(* IEC 61131-3 sources: ml2plc/benchmarks/st (part 17) *)

(* ---- MLP8_straton.st ---- *)
FUNCTION_BLOCK MLP8_FB

    (* Model Inputs/Outputs *)
VAR_INPUT
    input_data : REAL;
END_VAR

VAR_OUTPUT
    output_data : ARRAY[0..2] OF REAL;
END_VAR

VAR
    CONSTANT weights_0 : ARRAY[0..63] OF REAL := [0.566726267, 0.697450101, 0.648469865, -0.244775116, -0.237901151, 0.738550067, 0.472831041, 0.688409746, -0.0405910909, 0.54798907, 0.658046842, 0.487694085, 0.466130763, -0.209909201, -0.167861477, -0.185364306, -0.119988531, 0.702987075, 0.664516151, 0.492332131, 0.366119206, -0.231371135, 0.561849892, -0.299611568, 0.524393439, -0.0369002223, -0.225777417, 0.425555229, 0.708118021, 0.6373595, -0.302317858, 0.514846981, -0.277802587, -0.160284445, -0.23097758, 0.685079992, -0.0133622587, -0.197633862, 0.646109998, -0.0195143819, -0.00467607379, 0.46406725, -0.240666151, 0.522509336, -0.235457808, 0.497557789, -0.176456973, 0.530339539, -0.191211104, 0.541193664, 0.750494003, -0.0375860631, -0.214687645, -0.243620768, 0.659598589, 0.568989158, -0.3036699, 0.672104239, -0.244726226, 0.594575703, 0.681357145, -0.109698236, -0.107163459, 0.571734607];
    CONSTANT bias_0 : ARRAY[0..63] OF REAL := [-0.127067611, -0.150965586, -0.145847186, 0, 0, -0.142355159, 0.536983192, -0.151563853, 0, -0.108020559, 0.215985522, -0.109748609, -0.104939878, 0, 0, 0, 0, -0.15642038, -0.148533463, -0.110406905, 0.563737273, 0, -0.111798488, 0, -0.114780053, 0, 0, -0.0961699262, -0.133371383, -0.128657907, 0, -0.115175709, 0, 0, 0, -0.153447583, 0, 0, -0.0991757438, 0, 0, -0.103414647, 0, -0.117680125, 0, -0.111900046, 0, -0.119580522, 0, -0.121857166, -0.127358705, 0, 0, 0, -0.138788998, -0.125557691, 0, -0.147434101, 0, -0.126147434, -0.151844159, 0, 0, -0.126771837];
    CONSTANT weights_1 : ARRAY[0..3071] OF REAL := [-0.508529365, 0.777783334, -0.589114606, 0.647827327, -0.879598022, 0.374501675, -0.233010441, 0.470010132, 0.398335785, -0.835246623, -0.883157551, 0.755935609, -0.212538779, -0.178419977, 0.952007294, -0.811082065, 0.467197567, -0.294056267, -0.467858523, 1.01234376, 0.25377509, 0.712045431, -0.0497531593, -0.882072449, -0.987796485, 0.161702394, 0.587665379, 0.0541041195, 0.0643232763, 0.158115536, -0.557613134, -0.822882295, -0.602058291, -0.260582656, -1.05500817, -0.0198417753, 0.0395283103, 0.0372411311, 0.594341755, 0.584856927, 0.0607305169, -0.298460275, -0.480308563, 0.551810563, -0.737427711, 0.145618647, -0.499337137, -0.307826608, -0.473668456, 0.347774506, -0.187618226, 0.751432717, -0.689023435, 0.527891994, -0.193951294, 0.760585308, 0.328736782, -0.449620336, -0.498079717, 0.947781801, 0.0636215508, 0.190816671, 0.423609227, -0.963524342, 0.335212857, -0.300242186, -0.496480465, 0.62573868, 0.376674086, 0.36957857, 0.273251772, -0.723223269, -0.979038298, -0.128652185, 0.820281744, -0.150052547, -0.043580249, -0.184555292, -0.590572476, -1.00735581, -0.268060088, -0.245665103, -0.599425495, -0.135427296, -0.0110698044, -0.163606152, 0.57665354, 0.615970254, 0.0755210519, -0.242924631, -0.371946365, 0.521858156, -0.288352877, -0.214046448, -0.42009899, -0.499587744, -0.819006622, 0.522933841, -0.480003029, 0.688604951, -0.966424167, 0.622771263, -0.0291726999, 0.808974981, 0.633017004, -0.567950785, -0.715922832, 0.645944357, 0.126155347, 0.0951944366, 0.545724213, -0.931986749, 0.160165772, -0.0631896481, -0.52388972, 0.583337784, 0.470121413, 0.267368495, -0.0256699882, -1.1038264, -1.04683483, -0.0606382638, 0.849855661, 0.0996483564, -0.0824714303, 0.0362196565, -0.66673249, -1.04458475, -0.338297427, -0.53378427, -0.989768386, -0.225421071, 0.0280500948, 0.0889418721, 0.467521846, 0.709094465, 0.224540606, -0.255299211, -0.531706095, 0.613625348, -0.721871734, -0.14013961, -0.32255891, -0.276349634, -0.0558475852, -0.0150698572, 0.189445347, -0.224641621, 0.0600843728, -0.199145943, -0.114447266, 0.0321756005, -0.0139652044, 0.139568895, -0.136456579, 0.0218596458, 0.191010177, -0.0243975371, 0.0602264702, 0.0723614395, -0.0896188021, -0.058872506, 0.106127173, 0.0416764319, -0.0183494538, -0.199132025, 0.223530114, 0.00858539343, 0.0776902437, 0.0439737141, 0.00252109766, -0.226854458, 0.0800455809, 0.216010183, 0.174708903, -0.132116258, 0.0539589822, 0.0233850181, 0.126452208, 0.0195031166, 0.20596543, 0.0608135164, 0.0942558348, 0.22737518, -0.0990859717, -0.0777076781, -0.00981768966, -0.229763716, 0.0728095174, -0.208888695, -0.0588912666, 0.00719544291, -0.0642014891, 0.208572537, 0.185866833, -0.205061138, -0.190968722, -0.0123857558, 0.0851061344, 0.0569832623, 0.182903767, -0.165526241, -0.17117624, 0.0841451287, -0.178321734, -0.0988931656, 0.21516645, 0.203568548, -0.0786485076, 0.102775037, 0.104268342, 0.15373078, 0.23019889, 0.0220953524, -0.00975424051, 0.0953029096, -0.223771766, 0.229721338, -0.0257629901, 0.179429203, 0.0443455875, 0.191467524, 0.143349111, 0.21192956, 0.0171111971, -0.0315240026, 0.0892953277, -0.0647144169, -0.176158011, -0.0644855201, -0.15905486, -0.0899337977, 0.0437249541, 0.0412196219, -0.0510214269, -0.103800446, 0.0931487083, 0.183442682, 0.187456101, 0.18982622, -0.630144417, 0.611605942, -0.276451319, 0.63561976, -0.841786385, 0.105425507, 0.118410617, 0.642714441, 0.30139786, -0.423010617, -0.160331935, 0.631173253, -0.0531943738, 0.0132380854, 0.557571173, -0.680383444, 0.229302496, -0.0644649342, -0.597031713, 0.604079127, 0.0652358979, 0.508375168, 0.192985371, -0.684397638, -0.757217824, -0.0915823877, 0.624771178, 0.073392421, -0.213347048, -0.0439970493, -0.179815233, -0.822682321, -0.290968657, -0.449465156, -0.282994241, 0.0222680271, 0.202416599, 0.0366479158, 0.648888052, 0.345080584, -0.0183112063, -0.057644885, -0.33952108, 0.505236089, -0.269680262, 0.0832733512, -0.367935091, -0.27335614, 0.407757968, 0.238256618, 0.34742102, 0.0945411921, 0.179025948, -0.160453767, 0.0919690207, -0.0016620002, -0.140238672, 0.610232711, 0.662595987, 0.403355569, -0.108785428, 0.0517903045, 0.435860395, -0.0251670647, -0.251344532, 0.452141792, 0.557143986, 0.458476484, -0.255402505, 0.175111428, 0.455911607, 0.412472844, 0.218193471, -0.207911894, 0.0693136305, -0.059445411, -0.169521675, -0.182679832, 0.519502401, -0.0549139269, 0.497394502, 0.420575768, 0.255482435, -0.0491585582, 0.042904973, -0.192346439, 0.095114693, -0.346379042, -0.0267166235, 0.220421061, 0.3648085, -0.321888626, 0.446793377, -0.0310783982, 0.233682126, 0.388623834, -0.583991706, 0.505147576, -0.534565687, 0.322568089, -1.03081346, 0.283099979, 0.194360659, 0.706190765, 0.641339362, -0.426852167, -0.447203308, 0.554000199, 0.0497648604, 0.123939805, 0.853530824, -1.04427862, 0.252899885, -0.233157471, -0.306790262, 0.776063979, 0.559772849, 0.542160273, 0.0403436981, -1.10041475, -1.00884628, -0.138749599, 0.702059388, 0.0610145628, -0.0819382966, -0.111110725, -0.482868969, -0.934108913, -0.362628788, -0.359785378, -0.733438969, -0.060155347, -0.0659447312, 0.201255053, 0.359661549, 0.509634912, -0.0411985293, -0.504819214, -0.286087692, 0.544379532, -0.52835089, -0.0581299067, -0.380262613, -0.474460214, 0.0785628557, 0.193065852, -0.0540531427, 0.0867037475, -0.0140087456, -0.159107059, 0.16856578, 0.114497095, 0.0728079677, 0.123832315, 0.134191304, 0.201696187, -0.141746759, 0.213595003, -0.2263944, 0.0249090195, -0.158394754, -0.0716763884, 0.152066469, 0.0486070514, 0.111786395, 0.0807827115, 0.0409047008, 0.220125973, -0.219644442, 0.0905397534, 0.202887952, -0.153925478, -0.0712448508, 0.224727035, 0.116824895, 0.211984366, 0.0860830545, 0.134800911, -0.038962245, -0.0824456513, 0.0818852186, -0.0403479487, 0.0376374722, -0.108327284, 0.0718497038, 0.216866136, -0.213927254, 0.0031440109, -0.0106695592, -0.0465998203, -0.195866793, -0.214657992, -0.44059667, 0.660695314, -0.367561132, 0.594573438, -0.827821732, 0.38140139, -0.109366305, 0.564865768, 0.398382038, -0.642758369, -0.504486442, 0.811359286, 0.0293445885, -0.0519628488, 0.806313336, -0.863483965, 0.288089395, -0.143644974, -0.205591589, 0.838227034, 0.285395503, 0.240181088, 0.432383686, -0.649837255, -0.91485858, -0.177318007, 0.784425735, 0.22021389, 0.192846447, -0.0329939127, -0.348731846, -0.652700245, -0.339493215, -0.16938825, -0.534539282, 0.181898445, 0.178422064, -0.0549968779, 0.344090849, 0.254576117, -0.172308087, -0.139661431, -0.249803483, 0.395636946, -0.541676044, 0.201305479, -0.331647396, -0.306729645, 0.404410243, 0.250662118, 0.147280648, 0.502067685, 0.137784511, 0.0780866221, 0.0449218713, 0.323366255, 0.0272866227, 0.0769802928, -0.00688272109, 0.454549521, -0.147471949, -0.0136137269, 0.257623971, 0.0870388225, 0.0359390229, 0.164906204, 0.0806759894, 0.18752256, 0.211298063, 0.36549443, 0.381839573, 0.0227036048, 0.056207899, -0.0421615988, 0.497502565, 0.047046423, 0.209912181, 0.0365511775, 0.0822928399, 0.0565427281, 0.17033419, 0.133746162, -0.0657917038, -0.102406234, -0.0849392116, 0.171123147, 0.401582569, -0.0835181177, -0.133074522, 0.38805151, 0.281278849, 0.0756753385, 0.273700088, -0.114257708, 0.322280556, 0.240192294, -0.459217519, 0.901713192, -0.382146418, 0.67524451, -0.830624104, 0.424378633, -0.190720469, 0.905839324, 0.637098491, -0.503638327, -0.900598824, 1.19751096, 0.00358029734, -0.237770662, 1.01180136, -0.902854562, 0.475136936, -0.206849128, -0.774593174, 1.03993857, 0.640500665, 0.510213614, 0.0561259016, -1.24519598, -1.01733959, -0.115967944, 0.81452024, -0.161395952, -0.0437688082, -0.156050742, -0.53688693, -1.06002426, -0.470631003, -0.52531755, -1.12388718, 0.208761662, -0.176574588, -0.214394152, 0.646233439, 0.506878614, -0.0175239854, -0.63169241, -0.766251266, 0.681717753, -0.629178941, 0.117619962, -0.785952628, -0.735168219, -0.948679447, 0.878256857, -0.590300083, 1.04297566, -0.968591094, 0.856882274, 0.0444319323, 0.841967404, 0.672772825, -0.959409237, -0.734882236, 1.03502762, -0.0881304815, 0.137461543, 0.820007682, -1.38987863, 0.50563246, -0.212394595, -0.653115332, 1.03907979, 0.750977933, 0.649298608, -0.129806831, -1.40875912, -1.13032782, 0.180365622, 0.864530802, -0.155418515, -0.00242756307, -0.212027237, -0.488034099, -1.3115921, -0.619424522, -0.484913111, -1.09705448, -0.128922701, -0.13195011, -0.180079982, 1.18086195, 0.745139778, 0.167641819, -0.668225586, -0.77761519, 0.425894529, -0.626781106, -0.18818298, -0.721377492, -0.526926816, 0.215941429, -0.123659819, -0.184358388, 0.043376863, -0.0120955408, 0.122474253, -0.0583063215, -0.212231085, 0.183268249, 0.0962251723, -0.147334784, -0.11822731, 0.0362046957, 0.0269062817, -0.194129512, 0.0830053687, -0.161627054, -0.0567752719, -0.145187616, 0.120651454, -0.0233496577, 0.206467032, -0.17806983, -0.0681224167, 0.104563296, -0.218612805, 0.0865324736, 0.0349574983, -0.0137506574, 0.134827524, -0.0367743969, 0.184188545, 0.197318703, -0.0225695372, -0.221328974, -0.0929350406, -0.177381575, 0.00736005604, 0.037692219, 0.000573635101, 0.0186697245, -0.0238907337, -0.177731991, -0.129223391, 0.0824308693, -0.200551838, -0.16154848, 0.199765205, 0.206477582, 0.101242274, 0.0433039069, 0.0258513987, 0.160764426, -0.0691497177, -0.084734261, 0.227003336, -0.125068694, 0.146611392, -0.00917938352, -0.168416351, 0.136403561, -0.189610675, -0.127061039, 0.00317269564, 0.201314688, -0.0198562294, -0.144739896, 0.226294965, 0.228323668, 0.165590107, -0.173185229, -0.200818926, -0.0576947927, -0.000490188599, -0.104929939, -0.112846069, -0.00247612596, -0.132393166, -0.0162827373, -0.175804615, -0.149001211, 0.051792562, -0.14256072, -0.0560235083, -0.057627961, -0.214601696, -0.0697570592, -0.0851937234, -0.0509106219, 0.189388901, -0.223675087, 0.0777591765, -0.119579352, -0.0444692522, 0.196116835, -0.102969989, -0.184086397, -0.227760956, -0.0762356222, 0.193817228, -0.200928405, -0.101950482, 0.185671031, 0.192628652, 0.0269788206, 0.133608699, 0.033125788, 0.00712636113, 0.158508271, 0.222383291, 0.00950232148, -0.196249098, 0.0573975146, 0.177570045, -0.136008218, -0.0570820272, -0.149317741, 0.133439481, -0.10252957, -0.0730919391, -0.108708158, 0.0950632989, -0.000943243504, -0.192808211, 0.112221122, -0.227983013, 0.113385528, 0.0499848723, 0.07227844, -0.027736336, 0.0969584584, 0.0499704182, -0.015779078, 0.0496297777, -0.0482781082, -0.0640055835, 0.0741675794, 0.0220973194, 0.00619673729, 0.0708342195, 0.0922325552, 0.0812093318, 0.0475442708, 0.143843561, 0.0646075904, -0.120546937, 0.165627569, 0.0559816658, -0.207856715, -0.00720609725, -0.00766550004, -0.0709097236, 0.0499412119, -0.216208026, 0.101242423, 0.205707103, 0.0971380174, 0.17555812, 0.0319326222, 0.100855768, -0.0653036088, 0.170195639, -0.0348981768, 0.133284867, -0.165710002, 0.200018704, 0.0600594282, 0.16667527, -0.0698761344, 0.149929553, 0.164547354, 0.196463257, -0.0210942626, 0.150595009, 0.009890154, 0.165517092, -0.0509765595, 0.0195324123, -0.122422285, 0.0914077759, -0.0939736366, -0.043008998, -0.198219687, 0.0806815624, -0.116812088, -0.0638275146, 0.0568770766, -0.117142469, 0.229970008, 0.107616574, 0.0317450762, 0.173055828, -0.496262699, 0.528350115, -0.476345003, 0.706944287, -1.1584847, 0.553382933, -0.119421452, 0.475279957, 0.621614873, -0.557067633, -0.750136018, 0.550487518, 0.153488189, 0.0955926776, 0.441343844, -0.996506393, 0.396491706, -0.241655454, -0.664835751, 0.513887763, 0.287413418, 0.406024843, 0.181244105, -1.04969895, -1.03639233, -0.107004821, 0.723148108, -0.0915888399, 0.0190179348, 0.037515521, -0.378803849, -1.06744361, -0.268914074, -0.194677398, -0.675590158, -0.095566228, -0.159128696, 0.0355684161, 0.748913765, 0.683637083, 0.144258916, -0.341800094, -0.580741644, 0.453642994, -0.305999398, -0.210642919, -0.607958615, -0.411138088, -0.631047547, 0.31902054, -0.252779782, 0.601281404, -0.937315166, 0.595331609, -0.223486632, 0.800727427, 0.524395108, -0.632889867, -0.522368729, 0.613702238, 0.170364976, -0.0743942708, 0.881747961, -0.92249018, 0.504104912, -0.321216524, -0.560078859, 0.834637463, 0.195497125, 0.554065764, 0.00367344939, -1.11763585, -0.885221481, 0.0164854228, 0.888477564, -0.212700143, -0.0162799805, -0.0173875093, -0.256681591, -0.912996233, -0.589685977, -0.419041723, -0.830659449, 0.177183807, -0.023769334, 0.0620408952, 0.461648077, 0.596058011, -0.208506972, -0.514632285, -0.311666042, 0.440634817, -0.587510347, -0.0109222978, -0.662958026, -0.517027259, -0.837525904, 0.638323724, -0.36184296, 1.01570749, -0.784390688, 0.662208974, 0.0163894314, 0.649730861, 0.692022979, -0.625480831, -0.75872016, 0.904304087, -0.114221863, 0.0737056956, 0.882331848, -0.80644381, 0.392240912, -0.1903245, -0.660136998, 1.02926254, 0.28010729, 0.774872422, 0.0171470847, -1.19453144, -0.957866371, 0.0859950483, 0.974225044, -0.0765728354, -0.12548925, 0.098672539, -0.799499571, -0.906533301, -0.422217637, -0.347624362, -0.837638497, -0.225200176, -0.125213996, 0.0248761773, 0.615736663, 0.473281026, -0.0788344741, -0.188014746, -0.320240557, 0.684358001, -0.538594186, -0.148418903, -0.455669671, -0.77553618, 0.539408088, 0.166755497, 0.55472362, 0.265429348, 0.354455352, -0.276620895, -0.0783532336, 0.242457226, -0.41569528, 0.700103045, 0.649664283, 0.048536513, -0.158354238, -0.155874923, 0.300134778, 0.444611996, -0.0420008115, 0.55891937, 0.556732655, 0.0639907196, -0.266047776, 0.0416326076, 0.263084203, 0.212025434, 0.333977491, -0.161876708, 0.292763829, -0.129097462, -0.167351604, -0.0609775186, 0.47849986, 0.434941411, 0.452241063, 0.20276238, 0.156460658, -0.0998012573, -0.223118067, -0.101386949, 0.0894622728, -0.390977651, -0.165762499, 0.402601838, 0.58655256, -0.35624513, 0.586355329, -0.172513932, 0.670163631, 0.403929263, 0.111057967, -0.0854407847, 0.0988176763, 0.0290514529, -0.0514148921, 0.0591676235, -0.121268898, 0.0151776373, -0.164112777, -0.186199695, 0.152507097, -0.127331883, -0.0200016946, -0.218817249, -0.142015576, 0.0512357056, 0.1790497, 0.177341133, -0.171043411, -0.167235658, -0.184172481, 0.0341335535, 0.059614718, 0.183272332, 0.0454387665, 0.00863181055, -0.0723466873, -0.0487195253, 0.120217323, -0.0367092341, -0.0490668416, -0.0783792585, 0.0654979646, 0.0435450971, 0.0819463134, 0.164324373, -0.198321342, 0.153864235, 0.0049648881, 0.204122573, -0.14520669, -0.166048065, 0.15624702, 0.123243243, 0.026424855, 0.00905516744, 0.183895916, 0.0997058451, -0.430029929, 0.732694864, -0.38044247, 0.729891419, -0.619734049, 0.233270288, 0.133602768, 0.731909692, 0.346977323, -0.386733681, -0.66838181, 0.964729488, -0.252465546, -0.215632513, 0.727560103, -0.774502456, 0.215161905, 0.0859002024, -0.473885298, 0.682742119, 0.28458938, 0.447587937, 0.415456325, -0.487222195, -0.715709627, -0.173541993, 0.879550755, 0.110577703, -0.076938048, 0.10972473, -0.274036318, -0.707531929, -0.478892833, -0.0943468511, -0.363710195, 0.0505147278, 0.012673527, -0.00594107807, 0.703036904, 0.60320282, 0.181179851, -0.293641388, -0.339167327, 0.288456142, -0.319694757, -0.220214218, -0.521229386, -0.542298079, 0.157621264, 0.0535518527, 0.0709450841, 0.00566962361, -0.227724373, -0.123042539, -0.0993607342, -0.170529425, -0.188403592, 0.0198904574, 0.0604569316, -0.0971652716, -0.193837866, -0.115998521, -0.0477073491, 0.17740652, 0.0570174158, -0.0373788178, -0.116511613, 0.0726258159, -0.109403193, -0.0197265446, 0.198926538, -0.158025652, 0.191402584, 0.0438774228, -0.0633537173, -0.112080351, -0.207819521, 0.112972558, 0.172393352, -0.17403914, -0.0190575719, -0.188633874, 0.13436228, 0.00924527645, 0.0192586482, -0.0892033279, -0.198895514, -0.0415136367, 0.0746798813, -0.193610013, -0.0406213254, -0.0868264288, 0.181249648, 0.0303210616, 0.160136342, 0.055133611, -0.607501388, 0.728967071, -0.418366194, 0.571038365, -0.747898817, 0.22422646, -0.0210398231, 0.465642661, 0.310578942, -0.72168088, -0.809473634, 0.894424319, 0.0983128324, 0.107951425, 0.769080758, -0.861420989, 0.380020559, -0.0761527494, -0.688808799, 0.662312269, 0.276053041, 0.50488323, 0.188102454, -0.940027893, -1.04942298, 0.0129859298, 0.66093266, 0.126197129, -0.0100772232, -0.0683742166, -0.652829409, -0.910774648, -0.406400651, -0.246592462, -0.795169592, -0.173144892, 0.123221278, -0.0701487511, 0.638832688, 0.530133188, -0.218185201, -0.240693912, -0.617052913, 0.420573592, -0.416592866, -0.209370285, -0.289901704, -0.300533324, 0.188532501, -0.0149791986, 0.0226367414, -0.0932386518, 0.0710712969, 0.171038061, -0.164620638, -0.148197562, 0.145974845, -0.155826151, -0.150615975, -0.225483984, -0.11401882, 0.0688175559, 0.0625586808, -0.0694089085, -0.202945799, -0.0300859809, -0.151449189, -0.0992536247, -0.214120716, 0.231030732, 0.222256213, 0.181830227, -0.164005905, 0.223902106, -0.0978237242, -0.0618447214, -0.0550659746, -0.03302145, -0.0672846287, 0.126549751, 0.142029643, -0.159567744, -0.136364192, 0.11554879, 0.142483085, 0.222382694, 0.0213248134, 0.0888532102, 0.104086995, -0.168789625, -0.0168586224, -0.0982237905, 0.163628161, 0.049901545, -0.0885491371, 0.214760512, -0.0810971409, -0.0734869391, -0.10348469, 0.148927152, -0.0427333564, 0.157678753, -0.203982249, -0.13548547, -0.0630195141, 0.136405259, 0.0380123258, 0.0503391922, 0.104299515, 0.0854055583, 0.157218248, -0.0981568545, -0.0848319978, -0.0242888182, 0.225955576, 0.157761544, -0.0500846952, 0.122402251, 0.214099914, -0.166363984, -0.166297168, -0.201111734, 0.0539877415, -0.0838821232, 0.185279131, 0.0364579856, -0.0206628442, -0.0208719373, -0.1522457, -0.000124052167, 0.169354349, 0.064304024, -0.121528588, -0.137391984, -0.0628627986, 0.124056101, 0.158750266, -0.105839625, -0.110651106, -0.0281334817, 0.0249182284, -0.123197824, 0.198795587, -0.102469474, -0.883818984, 0.81256628, -0.796211541, 1.01723337, -1.29107821, 0.896784663, -0.161897063, 1.03797019, 0.619975567, -0.752187312, -0.861251831, 1.02046573, 0.107985839, -0.0928915367, 0.960325658, -1.24846256, 0.677723348, -0.626469016, -0.727811456, 1.10794473, 0.686511934, 0.562629521, -0.21034205, -1.16626048, -1.32185411, -0.0497885793, 1.41008556, 0.120183289, -0.15242587, -0.210768178, -0.786379874, -1.62433183, -0.901609361, -0.768333852, -1.33345139, -0.183859423, 0.191800296, 0.0267202556, 1.06132782, 0.971071541, 0.159037083, -0.778841496, -0.725091457, 0.797161579, -0.801008105, 0.0567008853, -0.926392496, -0.645901024, -0.569199502, 0.420701653, -0.428602308, 0.545880198, -0.542917073, 0.407910138, 0.0147776464, 0.492091984, 0.112967953, -0.519917846, -0.364893764, 0.711964726, -0.246900707, 0.174322069, 0.721634507, -0.438378364, 0.348643988, 0.249300689, -0.363233149, 0.518395662, 0.498299956, 0.495270997, 0.246642947, -0.824344754, -0.751605868, -0.0483377576, 0.759114742, -0.16243875, -0.0340996236, -0.196831778, -0.265718192, -0.494958758, -0.361495078, -0.128302455, -0.517697632, -0.188109025, 0.199257076, -0.0449238569, 0.503515899, 0.495425433, -0.223767415, 0.0430302434, -0.35435012, 0.17869848, -0.178660244, 0.182304084, -0.282319337, -0.294807643, -0.325249493, 0.68069011, -0.490325749, 0.485665023, -0.867332697, 0.273027927, -0.107890129, 0.543693006, 0.444793403, -0.601693988, -0.453863293, 0.880858183, -0.0925560892, -0.179236338, 0.631600976, -0.454414934, 0.212203413, 0.175340205, -0.466120481, 0.860624015, 0.1385369, 0.592696369, 0.0363957472, -0.8853392, -0.797631919, 0.0847206414, 0.532992899, -0.0990920961, -0.18515496, -0.00795261562, -0.16873166, -0.615779281, -0.384393632, -0.487988412, -0.676566958, 0.10417071, 0.00641438365, -0.00741529465, 0.464914918, 0.331140041, 0.0306460224, -0.232530951, -0.187347516, 0.408463717, -0.475631803, 0.118592083, -0.23730202, -0.434473544, 0.0895077288, -0.0349935293, -0.22308512, 0.0141319185, 0.0549576879, 0.0462970734, 0.20447138, -0.0055155009, -0.168662816, -0.204250544, -0.128070623, -0.166736096, 0.195838094, 0.0205055773, 0.0934391916, -0.160237819, 0.188507348, 0.225798249, 0.102597386, 0.211614758, -0.19942832, 0.212873966, -0.0228167474, -0.168969184, -0.0662842095, 0.0459339917, 0.178763598, 0.0424902141, -0.0532889664, -0.0481268018, 0.00563806295, -0.176516861, 0.114913225, 0.0826789737, 0.152797103, 0.160713494, 0.0820308328, 0.0364329815, -0.215456933, -0.0291685015, 0.00499258935, 0.172563821, 0.173846662, -0.130433768, -0.17989412, -0.193839312, -0.0669654459, 0.0631289482, -0.744850695, 0.645559728, -0.633206069, 0.704008698, -1.0611304, 0.654162765, 0.211175874, 0.915182769, 0.730826974, -0.480222166, -0.527996004, 0.89256072, 0.202866286, -0.206684694, 0.552212596, -1.02050734, 0.348888725, -0.249928072, -0.44374913, 1.0346396, 0.481733114, 0.506043792, -0.0193383321, -1.05336881, -1.26037169, -0.176632255, 1.03433955, 0.229603916, -0.0536026806, -0.0632608384, -0.376985997, -1.13252747, -0.83344084, -0.634874165, -0.963236511, -0.0154223144, 0.0877172351, -0.211326465, 0.92171514, 0.314691484, 0.0808647424, -0.427868694, -0.770184457, 0.296864182, -0.639095366, 0.106353432, -0.633490503, -0.714859784, -0.107103541, 0.101423919, 0.147723287, -0.164297104, 0.230882406, 0.0206960738, 0.0102013797, -0.0429925472, -0.077930674, -0.133540094, -0.110900417, -0.173496246, -0.0991988331, 0.0454862714, 0.18568024, -0.199032977, -0.0602819324, 0.180267125, 0.206567258, 0.205730617, 0.1114555, 0.173897982, -0.201017097, 0.130214989, -0.0398655385, -0.2129637, 0.0394511223, 0.116191447, -0.198193088, 0.0222576261, 0.182651192, -0.0370370746, 0.120660573, 0.0952059329, -0.14211534, 0.13360703, -0.161601901, -0.103214949, 0.00518859923, 0.183666885, -0.0247037411, -0.179946214, 0.116370827, -0.063356474, -0.120667845, 0.00735872984, -0.164149046, 0.208836943, -0.228432864, -0.183146626, -0.0760713965, 0.196719319, -0.219173297, -0.217832834, 0.0332981944, 0.0713680685, 0.0231516659, -0.20008482, -0.141936764, -0.0939454436, -0.0439056754, -0.0992506444, -0.0724140704, 0.00441415608, -0.0418925285, 0.091717422, 0.155868858, -0.187941268, 0.0954382122, -0.204097301, -0.0301216841, 0.177318573, -0.000473916531, 0.138970435, 0.0640658438, -0.0594422221, -0.169850349, -0.167840853, -0.130637288, 0.0395824611, 0.0593502223, -0.0275206268, -0.148664147, 0.0156640261, 0.109625578, 0.0748797655, -0.175359786, 0.0273132324, 0.0486470759, -0.147658646, -0.112167098, -0.198862731, -0.230632022, 0.168849111, 0.215680867, -0.0234110802, -0.0213709027, -0.0375050753, -0.0173404366, 0.0141991228, -0.149034426, -0.101356104, -0.0363372415, -0.0765377432, -0.0927268863, 0.132824361, 0.0599465966, 0.0326534808, 0.160957038, -0.10132587, -0.0343576521, 0.187982202, 0.170350194, 0.0885041654, 0.0257474184, 0.113371313, 0.153375179, 0.161880285, -0.00610806048, 0.16137439, 0.134935826, -0.188671395, 0.213962287, -0.201317504, 0.0826410651, -0.226450294, 0.216882646, -0.0690870732, 0.192525238, 0.212979048, 0.0936169922, -0.166921392, 0.0851119459, -0.00292879343, 0.134654909, 0.00792242587, -0.14447552, 0.10180673, 0.105806023, -0.163793385, -0.0397716165, 0.084336549, -0.0288007706, -0.0219024271, -0.788645625, 0.300676912, -0.434380859, 0.660915792, -1.05808699, 0.440583795, -0.0326454751, 0.377616823, 0.323617488, -0.759457648, -0.582121134, 0.743352175, 0.0626079515, -0.252789825, 0.828042924, -0.823172569, 0.481147766, -0.135181949, -0.743127644, 0.689704895, 0.494884163, 0.266731322, 0.236949638, -1.08205533, -0.981139362, -0.000693976879, 0.776560545, -0.00353519619, -0.181306928, -0.177135348, -0.639866769, -0.790730357, -0.507517576, -0.196227118, -0.64060837, 0.0397247672, -0.0699061602, 0.18094337, 0.518517315, 0.463519722, 0.206621543, -0.406967431, -0.428368241, 0.550414205, -0.460042566, -0.206967935, -0.661539197, -0.449288756, -0.160976678, 0.089292109, 0.182363629, -0.0687542707, 0.117252231, -0.0894444883, 0.097515285, 0.00596496463, -0.142512158, 0.109848678, -0.0957675427, 0.0741836429, -0.0711811632, -0.220404044, -0.0333378166, 0.0130293071, 0.167380124, -0.209830731, 0.0450258851, -0.216373578, -0.0252354294, -0.214120775, 0.0451754928, 0.0618753433, 0.124264568, 0.114782572, -0.0830270648, -0.0061095506, 0.0378096998, 0.193000734, 0.00110465288, -0.208948568, -0.227251396, 0.145473689, 0.0226551294, 0.0816588998, 0.142979681, 0.0730812848, 0.0112864524, 0.0950904489, 0.134623051, 0.229396313, 0.0646342337, 0.200954139, -0.183565915, -0.0515172482, 0.213664025, 0.0522184074, -0.130183578, -0.149197936, 0.190402538, -0.127790943, -0.129537612, -0.149094522, 0.0957980454, 0.203128397, 0.0133005232, -0.227951005, 0.144340754, 0.172468573, -0.128707811, -0.220882043, 0.0806925297, 0.10627833, -0.079099685, -0.151070029, 0.178314358, 0.0173286796, 0.0728730857, -0.0611997396, 0.177966416, -0.0243955404, -0.201305926, 0.0518709123, 0.0019980222, -0.0502954423, 0.0831291974, 0.0545895696, 0.192917913, -0.0607693791, 0.212297022, 0.209707111, -0.223003507, 0.157172948, 0.112241805, -0.13298136, -0.219473541, 0.017683953, 0.220878452, 0.155652612, -0.192422584, -0.185118213, -0.0381622612, -0.0616384, 0.213238835, -0.0145380646, -0.242232367, 0.183879182, -0.0200391226, 0.390113086, -0.529822767, 0.285439491, -0.0492200069, 0.630588651, 0.0329442956, -0.0533604547, -0.359910429, 0.815759659, 0.189301953, 0.0299578533, 0.553415775, -0.466774285, 0.423287809, 0.286925554, -0.406378478, 0.601928413, 0.133722708, 0.378852278, 0.263786614, -0.408895433, -0.327228457, -0.20093669, 0.429190964, -0.0700227022, -0.16383791, -0.115400337, -0.00653671892, -0.376550525, -0.249482572, -0.0984189957, -0.549010456, -0.207721353, -0.105499372, -0.18464458, 0.538136423, 0.233723909, 0.163720474, -0.0113063697, -0.0698213279, 0.0976555943, -0.287666231, -0.0449560732, -0.366864234, -0.0780268312, 0.154521793, -0.206957176, -0.00331628323, -0.0822689533, -0.141570732, -0.095661968, 0.190019131, -0.0730120391, -0.081034407, -0.0476873219, 0.152659744, -0.0459463447, -0.0765372962, -0.202615142, -0.151904061, -0.177600607, -0.0423512161, 0.165102661, 0.14116618, -0.163797587, -0.112091988, 0.133966058, 0.0903152227, 0.0881335437, 0.0512126982, -0.114689797, 0.0745567381, -0.0978981555, 0.184251398, -0.226357654, -0.0873684436, -0.147732317, 0.0203601718, -0.18398872, 0.0967339575, 0.221034557, 0.0497565866, 0.213030517, 0.0517413616, 0.145105839, 0.170207322, 0.192166746, -0.171817243, -0.187741011, 0.0901903808, 0.225754052, 0.141153336, 0.00577481091, -0.103353068, -0.074302271, -0.00892145932, -0.0783161372, -0.101536825, 0.0422692001, -0.199042976, 0.123941958, -0.152807683, -0.00614735484, -0.194417685, -0.184758469, 0.101321012, -0.121826246, -0.0651415884, -0.0327490717, 0.0212592781, 0.0575919747, -0.0404551774, -0.137311369, -0.0652063191, -0.193697706, -0.0827788562, 0.174635679, -0.193433821, -0.129116118, -0.199555337, -0.0278945416, -0.127540916, -0.0739758164, -0.227461636, 0.0502390563, 0.214967132, -0.180128664, -0.102538183, 0.200189888, 0.143446922, -0.19393146, 0.1378676, 0.0199711323, -0.0300057381, -0.166823938, 0.180752218, 0.0719076097, 0.126180381, -0.0845132619, 0.0907880962, 0.194829673, -0.663985848, 0.77064836, -0.374659657, 0.889753759, -0.975809515, 0.639838576, -0.126403913, 0.833601654, 0.654223442, -0.604557455, -0.877662063, 0.91747582, 0.148063019, -0.0108362213, 0.769826293, -1.03828716, 0.529056787, -0.184695244, -0.577510655, 1.0431757, 0.515663207, 0.543723166, 0.411439657, -1.07173824, -1.0059979, 0.190325856, 0.771367192, -0.0422332883, -0.154976666, -0.158998743, -0.552315474, -1.10934234, -0.806847394, -0.248423964, -0.91019249, 0.173593879, -0.0296967775, -0.100084677, 1.090855, 0.682509065, 0.0755710006, -0.463574976, -0.36591661, 0.361729652, -0.613674998, -0.105899826, -0.549840927, -0.62447834, -0.0463335663, -0.139898464, -0.19002527, 0.201583266, -0.0108013302, -0.143821821, -0.181311458, 0.00927944481, -0.176053047, 0.0897082686, 0.223907143, -0.0752439201, -0.17105864, -0.187036872, 0.196457207, -0.132100418, 0.0392292142, -0.225288749, 0.150229156, -0.208683252, 0.0060723573, -0.135761768, 0.123354644, 0.220038235, -0.0546040386, 0.13566041, 0.181121498, 0.0832488537, -0.10136041, 0.220071346, -0.00380316377, -0.179059088, 0.126896977, 0.0601697564, 0.155924767, -0.149190158, -0.0930504799, 0.180737764, -0.04751122, 0.0658206642, 0.0623811483, -0.120978415, 0.0224540234, 0.00235013664, -0.184219331, -0.00806756318, -0.116696037, -0.0770635903, -0.748862863, 0.691733062, -0.424329907, 0.799789727, -1.05946314, 0.298195779, 0.200020581, 0.586025238, 0.624388814, -0.658067703, -0.747551024, 1.04275012, -0.0187344868, 0.112926655, 0.976992071, -0.925199211, 0.607147694, -0.280815065, -0.695432901, 0.998307407, 0.462364107, 0.575792074, 0.172324777, -1.13321543, -0.905697048, 0.0550937355, 0.666969717, -0.0650874525, 0.0104155988, -0.137084335, -0.724511743, -0.795920372, -0.711852252, -0.451083243, -0.680145919, 0.208272308, 0.0677804053, -0.14033854, 0.735652745, 0.567496121, 0.0799567029, -0.218929842, -0.4710522, 0.543527842, -0.663609684, -0.228977308, -0.451376706, -0.715327144, 0.116782784, 0.205849856, 0.0496309698, 0.0113090724, -0.0841588229, -0.176505834, -0.222218573, -0.0656389594, -0.126934439, 0.132234335, -0.109233223, -0.0939592421, 0.157892436, -0.135368913, 0.11612004, -0.117877893, -0.0380255133, 0.187752604, -0.21574758, 0.174279958, -0.219665468, -0.0804129839, -0.0495111197, 0.182563394, 0.214952439, 0.132514298, -0.0940788239, 0.0368914902, 0.0827171504, 0.128636509, 0.156182349, 0.21208331, -0.141627356, -0.104670629, -0.12519595, -0.151801705, -0.22366339, -0.102302819, 0.0544782281, -0.185810149, 0.100636303, 0.102270424, 0.153328389, 0.152526736, -0.0473386198, 0.0830557644, -0.0707741976, -0.0522572547, -0.494424731, 0.736855507, -0.721928775, 0.594722331, -0.855316758, 0.616152048, 0.203238219, 0.625927567, 0.335482955, -0.811563671, -0.87894392, 1.06706297, 0.137062505, -0.0202609748, 0.959916353, -1.11030829, 0.608698785, -0.266370863, -0.477308273, 0.846952677, 0.624510765, 0.627845347, 0.0616629981, -1.34237301, -1.32277036, -0.00688707829, 0.872718215, 0.12940523, 0.10737741, -0.164741993, -0.769543707, -1.12598634, -0.479282528, -0.593654335, -0.804272413, 0.095541954, -0.13493672, -0.0239171684, 0.652407169, 0.673467875, -0.167755604, -0.452380717, -0.384234697, 0.665193677, -0.702400923, 0.196226805, -0.457769066, -0.418633968, 0.146774232, 0.113647103, 0.0468122661, -0.183789119, -0.0518778712, 0.0300752819, -0.218371764, 0.027431339, 0.102466434, -0.0275431871, 0.0386889279, 0.170658439, 0.0904044509, -0.200651497, 0.198548794, 0.0149045289, 0.118774742, -0.0857630968, 0.0440419018, 0.133314341, -0.0507946759, -0.0729796439, -0.0515012443, 0.0943579972, -0.126119778, 0.0275700092, 0.217315048, -0.0388335586, -0.168241814, -0.0159556717, -0.00677831471, 0.0058863312, -0.0642420501, 0.210292011, 0.0175138712, -0.0980680138, -0.0308899432, -0.199224621, -0.156486422, 0.157953531, 0.218261331, -0.139641479, 0.102292776, -0.17569083, 0.068279475, 0.109489173, -0.0230201036, -0.058723405, -0.496990621, 0.907003641, -0.544997454, 0.615387321, -0.907639384, 0.689036727, -0.10743545, 0.844478369, 0.397289991, -0.763743818, -0.761439562, 0.941512525, -0.0367905572, 0.176411226, 0.88902545, -0.766149938, 0.57171309, -0.191419542, -0.75722903, 0.796584249, 0.51507026, 0.595676959, 0.289120138, -0.851221859, -1.24790502, 0.00458748639, 0.989074171, -0.13295421, 0.0248681903, -0.033453539, -0.631120443, -0.808850586, -0.648837984, -0.685236216, -0.928007364, 0.154234052, 0.0611648262, 0.186276346, 0.623372674, 0.710519075, 0.0536311567, -0.219786227, -0.419961274, 0.388846785, -0.419767588, -0.0618833601, -0.753194571, -0.752672434, 0.0222598314, -0.103229627, 0.177644908, -0.0426572561, -0.0890138894, -0.00682736933, 0.155437946, -0.116798952, -0.117726527, 0.0264253616, -0.10268034, 0.0038767308, -0.0391207933, 0.211276978, -0.200906008, 0.00532445312, 0.126394689, 0.126339018, -0.0216406882, 0.0224532187, -0.0670201331, 0.171107739, 0.123936385, -0.0165472776, 0.222974986, 0.20747596, 0.141634315, 0.229873419, 0.197859794, 0.128305793, -0.0496525615, 0.0624574125, 0.00605608523, -0.0778746158, 0.0241027474, 0.0866435468, -0.189786866, 0.160087436, 0.202637553, -0.223458603, -0.0167357922, -0.188454032, 0.0181429535, -0.2130723, -0.022451669, 0.108265191, 0.218491733, 0.052171737, -0.652836621, 0.767383158, -0.42283994, 0.632724106, -1.13364995, 0.649288952, -0.0679906085, 0.527783275, 0.552915871, -0.81003809, -0.634466648, 1.0107944, 0.149907544, -0.0368661545, 0.781478763, -0.992297411, 0.624577761, -0.289075047, -0.745071769, 1.1118257, 0.316774637, 0.492890686, 0.0440929681, -1.07178032, -0.969130874, -0.15694207, 0.745540917, -0.142940223, -0.100186214, -0.0215469897, -0.373321265, -0.95797348, -0.464837581, -0.271017343, -0.847221971, 0.108970881, -0.0567243844, -0.108960621, 0.59346056, 0.712558091, 0.0655795336, -0.567239404, -0.283674717, 0.580327034, -0.447301775, 0.155937552, -0.793182433, -0.49744153, -0.238554373, 0.506624639, 0.00286697433, 0.598778844, -0.653696954, 0.309811443, -0.167876348, 0.311750382, 0.150085032, -0.284428507, -0.189132109, 0.590266764, -0.0625647008, 0.0517676473, 0.601453841, -0.310547978, 0.106867142, 0.265459538, -0.215828329, 0.591088116, 0.394775152, 0.161630541, 0.388673544, -0.68426609, -0.635585248, -0.080406189, 0.404845566, -0.134757608, 0.138952136, -0.212156534, -0.208190978, -0.357943833, -0.504545569, -0.334093183, -0.187557012, 0.209597796, -0.163752228, 0.0239533484, 0.499707729, 0.252578259, -0.145491198, -0.229706347, -0.278466046, 0.327976346, -0.283641189, 0.119131207, -0.281176746, -0.261819929, 0.00254940987, -0.108799152, 0.169640154, 0.0401595533, 0.152356386, -0.203051195, 0.0681574643, 0.00332997739, 0.134607494, -0.0376142859, 0.13674733, 0.139293373, -0.113252826, -0.119089492, -0.127502277, 0.151646078, 0.200112134, 0.0430138409, -0.215235919, -0.0758449733, 0.0214828551, 0.117211401, -0.0621953607, 0.13963601, -0.103949487, 0.0614436567, -0.148457155, -0.0485618562, -0.147884965, 0.0584875345, 0.0640005171, 0.132869005, 0.136009991, -0.0857912451, 0.0218506157, 0.124661952, 0.0290498734, 0.211057454, -0.170044988, 0.0348519981, -0.0899643153, 0.00265519321, 0.00405806303, 0.0331168473, 0.0907584429, -0.158105269, 0.117916793, 0.0351956189, -0.183738738, -0.182932615, -0.0161116123, -0.132023096, -0.140469611, 0.103275269, 0.107904017, 0.197627366, 0.0822747052, -0.0379109532, 0.0493098199, -0.0165452957, 0.0958584249, -0.0257950425, -0.0852105021, 0.213943928, 0.0791987777, -0.229539126, -0.0613196641, 0.162181169, -0.134439349, -0.142947942, 0.136250466, 0.177912503, -0.0891661942, -0.0219082683, 0.191606045, 0.203727961, -0.194567338, 0.178560197, -0.118050061, -0.0875838697, -0.032656461, -0.0749479234, 0.0135997236, 0.191686273, -0.0308628529, -0.107455276, -0.107913904, 0.123423457, 0.0380087495, -0.0611437857, -0.000918358564, 0.062859267, 0.166915208, -0.207877845, 0.0665597916, -0.0590146035, 0.0977552831, -0.0161778927, 0.153849542, 0.174365669, -0.0490427762, -0.141704723, -0.222182989, 0.087638557, -0.194510996, -0.213595271, -0.203084916, 0.0405931473, 0.107324213, -0.224449798, 0.12799567, -0.0140580833, -0.155599073, -0.212356359, 0.0655240715, 0.14629519, -0.0622795671, 0.171330899, -0.113621391, -0.163933933, 0.148270965, -0.189575627, 0.160233527, 0.0590209365, -0.0163397938, -0.158837885, -0.150075734, -0.0295645595, -0.0467994213, 0.138783991, 0.178417772, -0.216369763, -0.0769809186, -0.220601484, 0.116890937, 0.16154626, -0.182573706, 0.170100003, 0.110239148, 0.10367319, -0.131522372, -0.192169741, 0.19062677, -0.226928741, -0.49076128, 0.492487967, -0.377748668, 0.603053033, -0.918360233, 0.46039781, -0.127119377, 0.468201488, 0.560519755, -0.366247386, -0.774673104, 0.788756311, 0.0920332, -0.0813132748, 0.664744198, -0.849209249, 0.238996997, -0.189464867, -0.263247728, 0.811635613, 0.372185647, 0.429776549, 0.222558916, -0.708324492, -0.630015731, 0.0389983356, 0.827595592, -0.00504098833, -0.109677948, 0.0170855373, -0.559827507, -0.954249203, -0.290737808, -0.193426237, -0.731181085, -0.208241612, 0.229677647, -0.187462166, 0.44956404, 0.359694451, 0.0156254005, -0.244990766, -0.239677921, 0.385423601, -0.417864025, -0.202950597, -0.574585974, -0.238075972, -0.658879578, 0.652567625, -0.380847454, 0.536102772, -0.937951863, 0.545587242, 0.102139913, 0.494394481, 0.674190879, -0.707341909, -0.478948474, 1.0166322, -0.106750861, -0.209452301, 0.90282023, -0.734883547, 0.309125394, -0.0422016867, -0.437624246, 0.73226136, 0.377720475, 0.537338436, 0.223344579, -0.905140579, -1.05678511, -0.0109738857, 0.759665728, -0.150285929, 0.166756183, 0.104673982, -0.267434388, -1.0471257, -0.502471864, -0.197595, -0.875465453, -0.0973495841, -0.211485773, -0.00277207792, 0.797958732, 0.46998471, -0.231398359, -0.585462451, -0.586966991, 0.629688442, -0.568319738, 0.166556418, -0.646789789, -0.249907494, -0.0932250768, 0.199506938, -0.100093409, 0.149872005, 0.0996004939, -0.215020761, 0.221517682, 0.0143946409, -0.208271146, -0.173599541, -0.200193867, 0.11235258, -0.102700636, 0.128780276, 0.133931935, 0.0675489604, -0.143764541, -0.109202161, -0.0389329493, 0.065159291, 0.105982542, 0.0418533087, -0.201833695, -0.16808112, 0.051923722, -0.0987247974, 0.0472532511, -0.199569643, 0.0417475104, 0.207473457, -0.202503502, 0.0968965292, -0.166130066, -0.14273499, -0.104814321, 0.137824178, 0.107703924, 0.207627207, -0.0557606667, 0.126312077, 0.0482735336, 0.080401063, 0.0794066489, 0.186975449, -0.204078928, 0.121095777, 0.129890233, -0.200351194, -0.555514753, 0.440189064, -0.190514475, 0.782135725, -1.05458629, 0.190351352, 0.147283778, 0.766366899, 0.626958072, -0.59966433, -0.780890048, 0.8382864, -0.0354651734, 0.103119977, 0.510162055, -0.989340723, 0.386292875, -0.223132819, -0.43191573, 0.79997623, 0.584351182, 0.296678454, 0.301643163, -1.09266543, -0.904569089, 0.230082065, 0.620848179, -0.0371727198, -0.213054255, -0.181409121, -0.511923552, -0.685641944, -0.649093807, -0.252488911, -0.698802829, 0.108189613, -0.184165746, -0.154389888, 0.512973905, 0.664932311, -0.21917358, -0.292164713, -0.634630501, 0.381624997, -0.263713866, 0.160916567, -0.517369211, -0.385543734, -0.2176871, -0.220899865, 0.0958849192, 0.0384857953, 0.0021378994, 0.142900765, -0.0446970463, -0.156780541, 0.172815293, -0.104505956, 0.0622046292, 0.0989739001, 0.0780251026, -0.0743731856, -0.145816863, -0.217719108, -0.0956004411, -0.0359022319, -0.0968953669, 0.0927704275, 0.110802352, -0.168466851, -0.213452786, 0.126949996, 0.210244596, -0.181770414, 0.0876115263, -0.00970908999, 0.04316926, -0.0738278031, 0.175819457, 0.012167722, -0.143392116, 0.171328813, 0.155157655, -0.0616228282, 0.0531409085, -0.137051612, 0.228933036, -0.0683068484, -0.212712452, 0.0621427298, -0.0738676488, -0.171188653, -0.0592253506, 0.150956124, 0.162600875, -0.162026092, -0.582575023, 0.362777531, -0.174864829, 0.819940031, -0.803914487, 0.388996184, 0.0169635825, 0.545958996, 0.567325234, -0.561312914, -0.342158347, 0.948589146, -0.166090861, -0.0787301511, 0.606746793, -0.583138108, 0.269315422, 0.145984873, -0.468749732, 0.881489217, 0.158865809, 0.573085129, -0.0316874348, -0.926106632, -0.610725105, 0.138770849, 0.685023129, -0.0368995517, -0.0871459395, -0.0156094432, -0.511115313, -0.591342151, -0.316087872, -0.349807769, -0.814979374, -0.0717793554, 0.0488553643, 0.165656745, 0.777452707, 0.468234062, 0.117392659, -0.0483886674, -0.608514547, 0.492487013, -0.409540504, -0.176858068, -0.553234994, -0.465506107, -0.5408777, 0.727681696, -0.290462613, 0.52807337, -0.776279211, 0.251312613, 0.185282677, 0.796026111, 0.409259081, -0.6109429, -0.761808872, 0.647004008, 0.0717434138, -0.0945262313, 0.471209466, -0.793207943, 0.144436434, -0.0668516606, -0.635130227, 0.65240258, 0.553067803, 0.367429405, 0.228960067, -0.904923081, -0.812439024, -0.155557737, 0.832324028, -0.157464817, 0.00537765026, 0.0904373527, -0.477416456, -0.793419302, -0.726025105, -0.508038342, -0.646879554, 0.0079729706, -0.13128382, -0.203226566, 0.649361193, 0.39333272, 0.162937805, -0.267893493, -0.40245989, 0.462939024, -0.678447068, 0.00853562355, -0.524069667, -0.294732988, -0.0173678547, -0.173596948, 0.00478774309, 0.0496733189, 0.0307927728, -0.229844555, -0.215447322, -0.115677625, -0.215930954, -0.212037608, 0.121645361, 0.0949935317, -0.061223641, -0.00859671831, 0.0815468729, 0.0706126094, 0.141721606, -0.152815133, -0.00764629245, -0.157624185, -0.159587592, 0.157764137, 0.0981081426, 0.226554662, 0.17207396, 0.113308877, -0.169034466, 0.176956505, -0.18774581, -0.154347464, -0.15250954, 0.0999798477, 0.229934275, -0.0977487266, 0.153184742, -0.129915327, -0.0887184441, 0.18049556, -0.125426456, -0.175656229, -0.0141375959, 0.0338430703, -0.0391281843, 0.0500270426, 0.162896782, 0.0303710997, -0.151061252, -0.023189798, -0.0230622143, -0.0321559012, 0.0205596089, 0.106409997, -0.173725098, 0.11656481, -0.205545917, -0.187492684, 0.169136047, -0.230582356, -0.106434494, -0.120207116, 0.0903565586, 0.186642259, 0.0885660648, -0.208223954, 0.0594836175, 0.0968996286, 0.121583283, 0.200465769, 0.104577094, -0.0165389478, -0.0415070802, 0.181977838, 0.0383154452, -0.155830503, -0.153007895, 0.041195631, -0.186342672, -0.059953317, -0.0784820616, 0.154333293, -0.166642815, -0.209681675, 0.194542736, -0.0387383103, -0.166239113, -0.186846107, 0.133547276, -0.0147598982, 0.0936125219, 0.0422548056, -0.0737927109, -0.0658226013, -0.137619898, 0.0872041583, -0.117781766, -0.0487589687, -0.580934882, 0.533698261, -0.405752152, 0.697987616, -1.16385698, 0.32781446, -0.151206836, 0.747375369, 0.572708845, -0.612917125, -0.580609024, 0.757683396, -0.17346558, 0.158126444, 0.559633672, -1.0674212, 0.468338132, -0.149727091, -0.429316491, 0.661242127, 0.482864708, 0.59218806, 0.278764874, -1.14521229, -1.08595574, 0.0866391957, 0.885289967, 0.097596705, -0.0997715741, -0.169927061, -0.266317904, -1.02928007, -0.616001904, -0.245201156, -0.541648328, -0.0328267068, -0.120001011, -0.0568365157, 0.680588603, 0.611560047, -0.0473966859, -0.469011784, -0.565928638, 0.548262239, -0.462273121, 0.000132873654, -0.705312252, -0.563809395];
    CONSTANT bias_1 : ARRAY[0..47] OF REAL := [0.433181465, -0.159739494, 0.343099624, -0.0790926069, 0.242754415, -0.338606536, -0.0223293118, -0.185413241, -0.282873154, 0.401705146, 0.425327867, -0.139443144, 0.00381194474, -0.0179882385, -0.0181584675, 0.269541681, -0.317070097, 0.282907605, 0.377303362, -0.0464703776, -0.281575054, -0.21068567, 0.218524486, 0.278586447, 0.288027406, 0, -0.0332624279, 0, 0, 0, 0.341059655, 0.318366647, 0.461520761, 0.283488363, 0.236094803, 0, 0, 0, -0.107614197, -0.231008783, -0.00522471825, 0.342882812, 0.334155321, -0.239313349, 0.343503505, 0, 0.457686126, 0.335160881];
    CONSTANT weights_2 : ARRAY[0..143] OF REAL := [0.96770817, -0.0826222822, -1.67770183, -1.08297777, 0.190868899, 0.659189641, 0.52441889, 0.417532414, -1.1085583, -0.819571972, 0.534950435, 0.702221036, 1.33550215, -1.43372929, -0.135308087, -0.220515266, -1.13946176, 1.0897913, -0.326614529, -0.186647743, -0.0763737932, -0.631177902, 0.273417056, 0.735307574, -0.196904331, -1.43933821, 1.00949287, 0.81106329, 0.385401011, -1.15372264, 0.588859022, -0.166751906, -1.50449383, -0.973824382, 0.125834644, 0.377567172, -0.27398777, 0.004505869, -0.243019298, 0.247809455, 0.000650814385, 0.1305563, -0.900595546, 0.552432775, 0.379285604, 1.2473712, -1.12789369, -0.245032087, -0.370696455, -0.965937912, 1.10900915, -0.0585908629, 0.627174318, -0.782371938, 0.629469633, 0.0851785392, -1.57042968, -1.06669378, 0.362380683, 0.425719857, -0.507553756, -1.20341432, 1.01084483, -0.90987283, 0.0202404559, 0.734752774, -0.477947265, 0.378472954, -0.362295568, 1.15350997, -1.3812207, -0.323836356, 1.15531862, -1.29215503, -0.332708955, -0.202871636, -0.100203037, -0.101434514, -0.900261343, 0.471503556, 0.487855881, 0.126539111, 0.0417965055, -0.145941749, 0.203499347, -0.302549481, 0.336061329, -0.0208397806, 0.199737519, -0.0379016995, 0.536618233, 0.244431734, -1.25047731, 0.947521269, -1.58141315, -0.543069184, 0.391734958, 0.224103913, -0.980528355, 0.511248827, -0.000932945637, -2.0945518, 1.4905225, -1.63448358, -0.200654835, 0.128706932, 0.0916405022, 0.0111192763, -0.00716897845, -0.149395674, 0.209938854, 0.153475523, -0.288461208, 0.0753283799, -1.11330843, 0.111991018, 0.56435883, -0.0474135578, -1.5032984, 0.940999866, -0.300903082, 0.113724537, -0.210668802, 0.434426069, 0.549815357, -1.09440136, 0.741394579, 0.500292897, -1.21546543, 0.0351349264, -1.32852244, 1.02198708, 0.707758367, 0.410865933, -1.28819573, 0.287799746, -0.116568461, 0.217879742, 0.821959853, 0.50613308, -1.15333152, 0.714457929, 0.279045314, -1.1524899];
    CONSTANT bias_2 : ARRAY[0..2] OF REAL := [0.0925159603, 0.166509151, -0.274097234];
END_VAR

VAR
    (* Merged variables from all regions *)
    buffer_0 : ARRAY[0..47] OF REAL;
    buffer_1 : ARRAY[0..63] OF REAL;

    (* Temporary computation variables *)
    i : DINT;
    j : DINT;
    t : DINT;
    sum : REAL;
    (* Computation helpers *)
    max_val : REAL;
    exp_val : REAL;
    exp_sum : REAL;
    (* Spatial loop variables *)
    oc : DINT;
    oh : DINT;
    ow : DINT;
    ic : DINT;
    kh : DINT;
    kw : DINT;
    ih : DINT;
    iw : DINT;
END_VAR

(* Forward pass execution *)

(* Region: r0 [ACYCLIC] *)
(* Acyclic Region r0 *)
(* Layer 0: Fused Linear + RELU *)
FOR j := 0 TO 63 DO
    sum := 0.0;
    FOR i := 0 TO 0 DO
        sum := sum + input_data * weights_0[i * 64 + j];
    END_FOR;
buffer_1[j] := MAX(sum + bias_0[j], 0.0);
END_FOR;

(* Layer 1: Fused Linear + RELU *)
FOR j := 0 TO 47 DO
    sum := 0.0;
    FOR i := 0 TO 63 DO
        sum := sum + buffer_1[i] * weights_1[i * 48 + j];
    END_FOR;
buffer_0[j] := MAX(sum + bias_1[j], 0.0);
END_FOR;

(* Layer 2: Fused Linear + SOFTMAX *)
FOR j := 0 TO 2 DO
    sum := 0.0;
    FOR i := 0 TO 47 DO
        sum := sum + buffer_0[i] * weights_2[i * 3 + j];
    END_FOR;
output_data[j] := sum + bias_2[j];
END_FOR;

(* Softmax: find max *)
max_val := output_data[0];
FOR i := 1 TO 2 DO
    IF output_data[i] > max_val THEN
        max_val := output_data[i];
    END_IF;
END_FOR;

(* Softmax: compute exponentials and sum *)
exp_sum := 0.0;
FOR i := 0 TO 2 DO
    output_data[i] := EXP(output_data[i] - max_val);
    exp_sum := exp_sum + output_data[i];
END_FOR;

(* Softmax: normalize *)
FOR i := 0 TO 2 DO
    output_data[i] := output_data[i] / exp_sum;
END_FOR;

END_FUNCTION_BLOCK
